{attribute 'GeneratedUsingTerminal: EK1100-0000-0018'}
{attribute addProperty BoxType "EK1100-0000-0018"}
{attribute addProperty Id "Beckhoff_EL19xxEK1122Beckhoff_EL19xxEK1122_2AE5B5792A_0001_EL1918_0000_0016EL1918_D38ABFDC40"}
{attribute addProperty CRC "1292584276"}
{attribute addProperty Size "42"}
TYPE Beckhoff_EL19xx_4D0B4554 EXTENDS EK1100_1FC0878B :
STRUCT
	{attribute addProperty Name "Beckhoff_EL19xxEK1122"}
	{attribute addProperty PreviousPort "Beckhoff EL19xx : B"}
	Beckhoff_EL19xxEK1122 : Beckhoff_EL19xxEK1122_2AE5B579;
	{attribute addProperty Name "A_0001_EL1918_0000_0016"}
	{attribute addProperty PreviousPort "Beckhoff EL19xxEK1122 : C"}
	A_0001_EL1918_0000_0016 : EL1918_D38ABFDC;
END_STRUCT
END_TYPE

(* stored: Version 1.2.0.0, ProductVersion 3.1.4024.9
   DUT Beckhoff_EL19xx_4D0B4554: Id {ee222906-6b95-41e8-9127-a2f6dad08cbf} *)
